TYPE TrayLoad_Outputs_typ:
STRUCT
	BallClampOpen AT %Q*: BOOL;
	BallClampClose AT %Q*: BOOL;
	LoadTray AT %Q*: BOOL;
END_STRUCT
END_TYPE

(* stored: Version 1.1.0.1, ProductVersion 3.1.4024.12
   DUT TrayLoad_Outputs_typ: Id {65939ab6-81f5-0d36-388e-603677745237} *)
